// TIA Portal V18 export
// export: Created 2026-01-09T11:31:59.0829608Z, ExportSetting WithDefaults, DisplayName Totally Integrated Automation Portal, DisplayVersion V18 Update 5, DisplayName TIA Portal Openness, DisplayVersion V18 Update 5, DisplayName TIA Portal Teamcenter Gateway, DisplayVersion V18, DisplayName TIA Portal Version Control Interface, DisplayVersion V18, DisplayName SINAMICS Startdrive Advanced, DisplayVersion V18 SP2 Update 1, DisplayName SINAMICS Startdrive G110M, G120, G120C, G120D, G120P, G115D, DisplayVersion V18 SP2 Update 1, DisplayName SINAMICS Startdrive G130, G150, S120, S150, SINAMICS MV, S210, G220, S200, DisplayVersion V18 SP2 Update 1, DisplayName STEP 7 Professional, DisplayVersion V18 Update 5, DisplayName STEP 7 Safety, DisplayVersion V18, DisplayName WinCC Professional, DisplayVersion V18 Update 5
TagTable "TipWord"
  GlobalTip_01 : Word  (%DB1069.DBW0, CPU S71500-2PN_TP700, 100 ms)
  GlobalTip_02 : Word  (%DB1069.DBW2, CPU S71500-2PN_TP700, 100 ms)
  GlobalTip_03 : Word  (%DB1069.DBW4, CPU S71500-2PN_TP700, 100 ms)
  GlobalTip_04 : Word  (%DB1069.DBW6, CPU S71500-2PN_TP700, 100 ms)
  GlobalTip_05 : Word  (%DB1069.DBW8, CPU S71500-2PN_TP700, 100 ms)
  GlobalTip_06 : Word  (%DB1069.DBW10, CPU S71500-2PN_TP700, 100 ms)
  GlobalTip_07 : Word  (%DB1069.DBW12, CPU S71500-2PN_TP700, 100 ms)
  GlobalTip_08 : Word  (%DB1069.DBW14, CPU S71500-2PN_TP700, 100 ms)
  GlobalTip_09 : Word  (%DB1069.DBW16, CPU S71500-2PN_TP700, 100 ms)
  GlobalTip_10 : Word  (%DB1069.DBW18, CPU S71500-2PN_TP700, 100 ms)
  GlobalTip_OP1 : Word  (%DB1069.DBW20, CPU S71500-2PN_TP700, 100 ms)
  GlobalTip_OP2 : Word  (%DB1069.DBW22, CPU S71500-2PN_TP700, 100 ms)
